# EPICS IOC start-up script: test/startup/st.mcu035-PTP-B02.iocsh
epicsEnvSet("MOTOR_PORT",    "$(SM_MOTOR_PORT=MCU1)")
epicsEnvSet("IPADDR",        "$(SM_IPADDR=172.30.38.73)")
epicsEnvSet("IPPORT",        "$(SM_IPPORT=48898)")
epicsEnvSet("AMSNETIDIOC",   "$(SM_AMSNETID=172.30.38.12.1.1)")
epicsEnvSet("ASYN_PORT",     "$(SM_ASYN_PORT=MC_CPU1)")
epicsEnvSet("PREFIX",        "$(SM_PREFIX=LabS-MCAG:MC-MCU-035:)")
epicsEnvSet("PREC",          "$(SM_PREC=3)")
epicsEnvSet("SM_NOAXES",     "1")
epicsEnvSet("ECM_OPTIONS",   "adsPort=852;amsNetIdRemote=5.36.136.2.1.1;amsNetIdLocal=$(AMSNETIDIOC)"

# Do not start the poller yet
epicsEnvSet("ECM_MOVINGPOLLPERIOD", "0")
epicsEnvSet("ECM_IDLEPOLLPERIOD",   "0")

< ethercatmcController.iocsh
< ethercatmcEL6688-PTP.iocsh
< ethercatmcEL6688-EL1252-PTP.iocsh

#####################################################
# EL1252, first channel, CHNO == 0
epicsEnvSet("CHNO",     "0")
< ethercatmcEL1252-OneChannel.iocsh

#####################################################
# PTP with ExtSync
< ethercatmcEL6688-PTP.iocsh

#
# Start polling, values are in millisconds
#
epicsEnvSet("MOVINGPOLLPERIOD", "500")
epicsEnvSet("IDLEPOLLPERIOD",   "500")
ethercatmcStartPoller("$(MOTOR_PORT)", "$(MOVINGPOLLPERIOD)", "$(IDLEPOLLPERIOD)")
